TYPE TcoInsightCommandControl_v_5_x_x : 
STRUCT
    CurrentJobID AT %I* : UINT;
    Command AT %Q* : UINT;
END_STRUCT
END_TYPE

(* stored: Version 1.1.0.1, ProductVersion 3.1.4024.11
   DUT TcoInsightCommandControl_v_5_x_x: Id {c61b9e66-a143-0653-0650-6fb98a4d9c64} *)
